FUNCTION_BLOCK AccelDecel (* Basic Function Block Type *)
  (* Standard: 61499-2 *)
  (* Version 0.2, 2003-12-04, JHC, Rockwell Automation, Renamed for better indexing. *)
  (* Version 0.1, 2002-11-05, JHC, Rockwell Automation, Corrected missing ST element in Algorithm REQ. *)
  (* Version 0.0, 2000-05-30, JHC, Rockwell Automation *)
  (* Compiler header: package fb.rt.benchmarks.cruisecontrol; *)
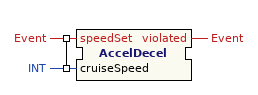
  EVENT_INPUT
    speedSet WITH cruiseSpeed;
  END_EVENT
  EVENT_OUTPUT
    violated; (* Initialization Confirm *)
  END_EVENT
  VAR_INPUT
    cruiseSpeed : INT; (* Input event qualifier *)
  END_VAR
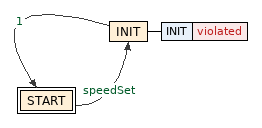
  EC_STATES
    START; (* Initial State *)
    INIT : INIT -> violated; (* Initialization *)
  END_STATES
  EC_TRANSITIONS
    START TO INIT := speedSet;
    INIT TO START := 1;
  END_TRANSITIONS
  ALGORITHM INIT IN ST: (* Initialization algorithm *)

  END_ALGORITHM
END_FUNCTION_BLOCK
